KUKA KRL program: chk_w4_grp1_clo.src

&ACCESS RVO2
&COMMENT Check GRP ACCELO Z1 CLOSE
DEF chk_w4_grp1_clo( )

;//---- Start User-------
;Aguardando posicao de gripper fechado

$TIMER[10] = 0
$TIMER_STOP[10] = FALSE

WAIT FOR (NOT $IN[37] AND NOT $IN[39])
WAIT FOR ($IN[38] AND $IN[40])

$TIMER_STOP[10] = TRUE
$TIMER[10] = 0

;//---- End User-------

END
